FUNCTION_BLOCK AE_MERGE_3 (* MERGE 3 AE into 1 AE (generic FB) *)
  (* Standard: 61499-2; Description: Copyright (c) 2026 Meisterschulen am Ostbahnhof This program and the accompanying materials are made available under the terms of the Eclipse Public License 2.0 which is available at https://www.eclipse.org/legal/epl-2.0/ SPDX-License-Identifier: EPL-2.0 *)
  (* Version 1.0, 2026-09-06, Franz Höpfinger, Meisterschulen am Ostbahnhof *)
  PACKAGE adapter::events::unidirectional;
  IMPORT eclipse4diac::core::GenericClassName;
  {SET_ATTRIBUTE(eclipse4diac::core::GenericClassName, 'GEN_AE_MERGE')}
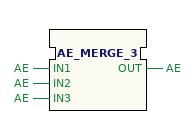
  SOCKETS
    IN1 : adapter::types::unidirectional::AE;
    IN2 : adapter::types::unidirectional::AE;
    IN3 : adapter::types::unidirectional::AE;
  END_SOCKETS
  PLUGS
    OUT : adapter::types::unidirectional::AE;
  END_PLUGS
END_FUNCTION_BLOCK
